(* CoDeSys 2.3.9.35 project: PROJETO_MAQUINA_ESTADO.pro *)
(* Author: João Marangoni *)
(* Libraries: SysLibTargetVisu.lib 26.11.08 09:50:36, Standard.lib 26.11.08 09:46:20, Iecsfc.lib 26.11.08 09:46:14, DU35x.lib 26.11.09 14:36:14, SYSLIBCALLBACK.LIB 26.11.08 09:50:38 *)

(* PLC configuration (modules and I/O channels)
Communication [Comunica] node 0, in %IB0 out %QB0
  COM1 [COM1] node 0, in %IB0 out %QB0 {BaudRate = 115200; Paridade = No Parity; StopBits = 1 Stop Bit; Modem = Without RTS/CTS; Delay = 5}
    MToolIEC [Codesys] node 0, in %IB0 out %QB0
  COM2 [COM2] node 1, in %IB0 out %QB0 {BaudRate = 115200; Paridade = No Parity; StopBits = 1 Stop Bit; Modem = Without RTS/CTS; Delay = 5}
    Disable [Desabilitado485] node 0, in %IB0 out %QB0
BOTAO_LIGA AT %IX0.0 [BitInput] I0.0
BOTAO_DESLIGA AT %IX0.1 [BitInput] I0.1
SENSOR_NIVEL_ALTO AT %IX0.2 [BitInput] I0.2
SENSOR_NIVEL_BAIXO AT %IX0.3 [BitInput] I0.3
I04 AT %IX0.4 [BitInput] I0.4
I05 AT %IX0.5 [BitInput] I0.5
I06 AT %IX0.6 [BitInput] I0.6
I07 AT %IX0.7 [BitInput] I0.7
I08 AT %IX0.8 [BitInput] I0.8
Digital Inputs 1 [Entradas1] node 0, in %IW1 out %QB0
  I10 AT %IX1.0 [BitInput] I1.0
  I11 AT %IX1.1 [BitInput] I1.1
  I12 AT %IX1.2 [BitInput] I1.2
  I13 AT %IX1.3 [BitInput] I1.3
  I14 AT %IX1.4 [BitInput] I1.4
  I15 AT %IX1.5 [BitInput] I1.5
  I16 AT %IX1.6 [BitInput] I1.6
  I17 AT %IX1.7 [BitInput] I1.7
  I18 AT %IX1.8 [BitInput] I1.8
Digital Inputs 2 [Entradas2] node 0, in %IW2 out %QB0
  I20 AT %IX2.0 [BitInput] I2.0
  I21 AT %IX2.1 [BitInput] I2.1
Analog Inputs [EntradaAnalogica] node 0, in %IW4 out %QB0
  AI0 AT %IW4 [WordInput] AI0 {TipoAnalogica = Channel Disable; FiltroAnalogica = Filter 0 - AI=2ms  / AV=90ms; FundoEscala = 0}
  AI1 AT %IW5 [WordInput] AI1 {TipoAnalogica = Channel Disable; FiltroAnalogica = Filter 0 - AI=2ms  / AV=90ms; FundoEscala = 0}
  AI2 AT %IW6 [WordInput] AI2 {TipoAnalogica = Channel Disable; FiltroAnalogica = Filter 0 - AI=2ms  / AV=90ms; FundoEscala = 0}
  AI3 AT %IW7 [WordInput] AI3 {TipoAnalogica = Channel Disable; FiltroAnalogica = Filter 0 - AI=2ms  / AV=90ms; FundoEscala = 0}
Fast Inputs [EntradasRapidas] node 1, in %IB16 out %QB0
  Block 0 [Bloco0] node 0, in %IB16 out %QB0
    Disable [DesabilitadoBloco0] node 0, in %IB16 out %QB0
  Block 1 [Bloco1] node 1, in %IB16 out %QB0
    Disable [DesabilitadoBloco1] node 0, in %IB16 out %QB0
  Configurable Input Block 0 [EntradaConfiBloco0] node 2, in %IB16 out %QB0
    Counter 0 [EntradaConfContador0] node 0, in %IB16 out %QB0 {EntradaConfiguravelContador = Disable}
  Configurable Input Block 1 [EntradaConfiBloco1] node 3, in %IB16 out %QB0
    Counter 2 [EntradaConfContador2] node 0, in %IB16 out %QB0 {EntradaConfiguravelContador = Disable}
MOTOR_AGITO AT %QX0.0 [BitOutput] Q0.0
VALVULA_ENTRADA1 AT %QX0.1 [BitOutput] Q0.1
VALVULA_ENTRADA2 AT %QX0.2 [BitOutput] Q0.2
VALVULA_SAIDA AT %QX0.3 [BitOutput] Q0.3
Q04 AT %QX0.4 [BitOutput] Q0.4
Q05 AT %QX0.5 [BitOutput] Q0.5
Q06 AT %QX0.6 [BitOutput] Q0.6
Q07 AT %QX0.7 [BitOutput] Q0.7
Digital Outputs 1 [Saidas1] node 0, in %IW0 out %QW1
  Q10 AT %QX1.0 [BitOutput] Q1.0
  Q11 AT %QX1.1 [BitOutput] Q1.1
  Q12 AT %QX1.2 [BitOutput] Q1.2
  Q13 AT %QX1.3 [BitOutput] Q1.3
  Q14 AT %QX1.4 [BitOutput] Q1.4
  Q15 AT %QX1.5 [BitOutput] Q1.5
  Q16 AT %QX1.6 [BitOutput] Q1.6
  Q17 AT %QX1.7 [BitOutput] Q1.7
Analog Outputs [SaidaAnalogica] node 0, in %IW0 out %QW3
  AO0 AT %QW3 [WordOutput] AO0 {TipoAnalogica = Channel Disable; FundoEscala = 0}
  AO1 AT %QW4 [WordOutput] AO1 {TipoAnalogica = Channel Disable; FundoEscala = 0}
Fast Outputs [SaidasRapidas] node 1, in %IB0 out %QB10
  Fast Output 0 Disable [DesabilitadoF0] node 0, in %IB0 out %QB10
  Fast Output 1 Disable [DesabilitadoF1] node 1, in %IB0 out %QB10
Counter Output [SaidasContador] node 2, in %IB0 out %QB10
  Block 0 Output Disable [DesabilitadoSaidaBloco0] node 0, in %IB0 out %QB10
  Block 1 Output Disable [DesabilitadoSaidaBloco1] node 1, in %IB0 out %QB10
External Events [Eventos] node 2, in %IB13 out %QB6
  Timer Event [TimerEvent] node 0, in %IB13 out %QB6 {Intervalo = 10}
*)

(* Global variable list: Variáveis globais *)
VAR_GLOBAL
	ABASTECIMENTO: BOOL;
	TIMER_AGITO: TON;
	Count_On: TIME;
END_VAR

(* POU PLC_PRG, LD *)
PROGRAM PLC_PRG
VAR
END_VAR
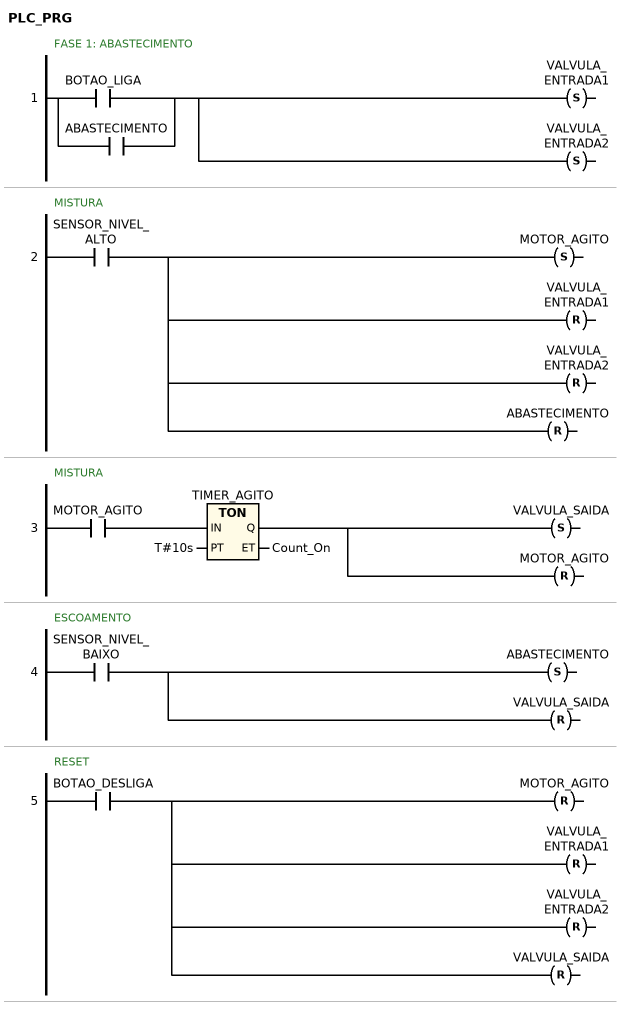
_LD_ (* Ladder Diagram *)
NETWORK 1 (* FASE 1: ABASTECIMENTO *)
	{ [BOTAO_LIGA] | [ABASTECIMENTO] } --- (S VALVULA_ENTRADA1) (S VALVULA_ENTRADA2)
NETWORK 2 (* MISTURA *)
	[SENSOR_NIVEL_ALTO] --- (S MOTOR_AGITO) (R VALVULA_ENTRADA1) (R VALVULA_ENTRADA2) (R ABASTECIMENTO)
NETWORK 3 (* MISTURA *)
	[MOTOR_AGITO] - TIMER_AGITO:TON(IN: *, PT: T#10s, ET => Count_On) --- (S VALVULA_SAIDA) (R MOTOR_AGITO)
NETWORK 4 (* ESCOAMENTO *)
	[SENSOR_NIVEL_BAIXO] --- (S ABASTECIMENTO) (R VALVULA_SAIDA)
NETWORK 5 (* RESET *)
	[BOTAO_DESLIGA] --- (R MOTOR_AGITO) (R VALVULA_ENTRADA1) (R VALVULA_ENTRADA2) (R VALVULA_SAIDA)
_END_LD_
(* the same logic as Structured Text *)
(* Network 1: FASE 1: ABASTECIMENTO *)
IF BOTAO_LIGA OR ABASTECIMENTO THEN VALVULA_ENTRADA1 := TRUE; VALVULA_ENTRADA2 := TRUE; END_IF;
(* Network 2: MISTURA *)
IF SENSOR_NIVEL_ALTO THEN MOTOR_AGITO := TRUE; VALVULA_ENTRADA1 := FALSE; VALVULA_ENTRADA2 := FALSE; ABASTECIMENTO := FALSE; END_IF;
(* Network 3: MISTURA *)
TIMER_AGITO(IN := MOTOR_AGITO, PT := T#10s);
Count_On := TIMER_AGITO.ET;
IF TIMER_AGITO.Q THEN VALVULA_SAIDA := TRUE; MOTOR_AGITO := FALSE; END_IF;
(* Network 4: ESCOAMENTO *)
IF SENSOR_NIVEL_BAIXO THEN ABASTECIMENTO := TRUE; VALVULA_SAIDA := FALSE; END_IF;
(* Network 5: RESET *)
IF BOTAO_DESLIGA THEN MOTOR_AGITO := FALSE; VALVULA_ENTRADA1 := FALSE; VALVULA_ENTRADA2 := FALSE; VALVULA_SAIDA := FALSE; END_IF;
END_PROGRAM

(* Visualisation NEWVISUALIZACION
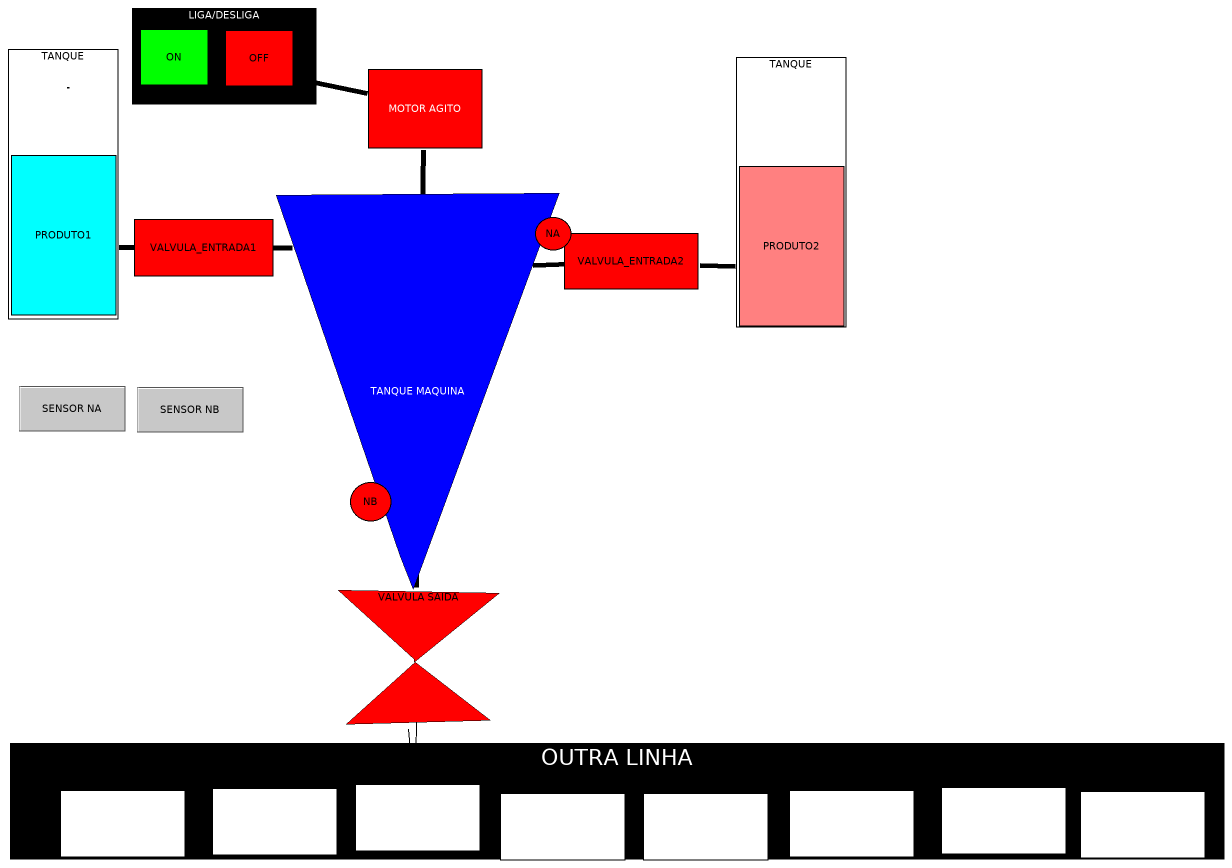
rectangle at (86,57)-(196,327): text "TANQUE"
rectangle at (89,163)-(194,323): text "PRODUTO1"
rectangle at (210,16)-(394,112): text "LIGA/DESLIGA"
rounded rectangle at (446,77)-(560,156): text "MOTOR AGITO"; alarm colour if .MOTOR_AGITO
polygon at (416,598)-(577,670): text "VALVULA SAIDA"; alarm colour if .VALVULA_SAIDA
polygon at (424,670)-(568,732): alarm colour if .VALVULA_SAIDA
polygon at (354,201)-(637,597): text "TANQUE MAQUINA"
rounded rectangle at (212,227)-(351,284): text "VALVULA_ENTRADA1"; alarm colour if .VALVULA_ENTRADA1
rounded rectangle at (642,241)-(776,297): text "VALVULA_ENTRADA2"; alarm colour if .VALVULA_ENTRADA2
rectangle at (814,65)-(924,335): text "TANQUE"
rectangle at (817,174)-(922,334): text "PRODUTO2"
ellipse at (613,225)-(649,258): text "NA"; alarm colour if .SENSOR_NIVEL_ALTO
ellipse at (428,490)-(469,529): text "NB"; alarm colour if .SENSOR_NIVEL_BAIXO
rounded rectangle at (88,751)-(1302,867): text "OUTRA LINHA"
rounded rectangle at (218,37)-(286,93): text "ON"; taps .BOTAO_LIGA
rounded rectangle at (303,38)-(371,94): text "OFF"; taps .BOTAO_DESLIGA
button at (97,394)-(203,439): text "SENSOR NA"; toggles .SENSOR_NIVEL_ALTO
button at (215,395)-(321,440): text "SENSOR NB"; toggles .SENSOR_NIVEL_BAIXO
17 more shapes without text or variables
*)
